// TIA Portal V17 export
// export: Created 2023-02-26T22:59:49.7304626Z, ExportSetting WithDefaults, DisplayName Totally Integrated Automation Portal, DisplayVersion V17, DisplayName TIA Portal Openness, DisplayVersion V17, DisplayName TIA Portal Version Control Interface, DisplayVersion V17, DisplayName TIA Portal Test Suite Advanced, DisplayVersion V17, DisplayName STEP 7 Professional, DisplayVersion V17, DisplayName SIMATIC Energy Suite, DisplayVersion V17, DisplayName STEP 7 Safety, DisplayVersion V17, DisplayName WinCC Professional, DisplayVersion V17
FUNCTION "LOG_ModeTime" : Void   // FC18, LAD
{ S7_Optimized_Access := 'TRUE' }
VERSION : 0.1
// stored: AutoNumber true, IsIECCheckEnabled false, SetENOAutomatically false, UDAEnableTagReadback false
   VAR_TEMP
      t_RisingEdge : Bool;
   END_VAR
BEGIN

REGION Network 1: Trigger
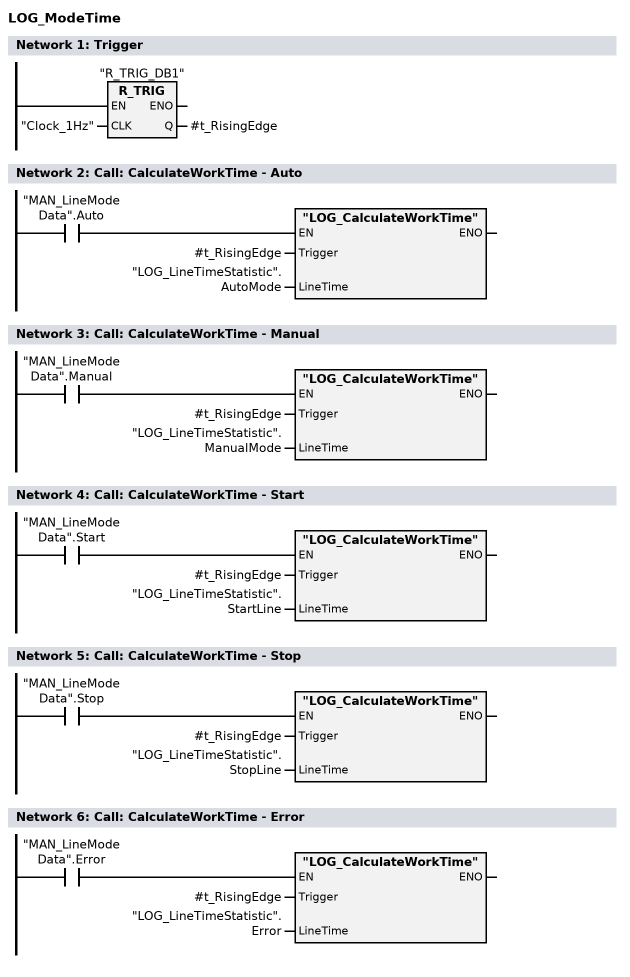
   RUNG wire#powerrail
      "R_TRIG_DB1".R_TRIG(CLK := "Clock_1Hz", Q => #t_RisingEdge)
   END_RUNG
   // the same network as SCL:
   "R_TRIG_DB1"(CLK := "Clock_1Hz", Q => #t_RisingEdge);   // R_TRIG
END_REGION

REGION Network 2: Call: CalculateWorkTime - Auto
   RUNG wire#powerrail
      Contact( "MAN_LineModeData".Auto )
      "LOG_CalculateWorkTime"(Trigger := #t_RisingEdge, LineTime := "LOG_LineTimeStatistic".AutoMode)
   END_RUNG
   // the same network as SCL:
   IF "MAN_LineModeData".Auto THEN
       "LOG_CalculateWorkTime"(Trigger := #t_RisingEdge, LineTime := "LOG_LineTimeStatistic".AutoMode);
   END_IF;
END_REGION

REGION Network 3: Call: CalculateWorkTime - Manual
   RUNG wire#powerrail
      Contact( "MAN_LineModeData".Manual )
      "LOG_CalculateWorkTime"(Trigger := #t_RisingEdge, LineTime := "LOG_LineTimeStatistic".ManualMode)
   END_RUNG
   // the same network as SCL:
   IF "MAN_LineModeData".Manual THEN
       "LOG_CalculateWorkTime"(Trigger := #t_RisingEdge, LineTime := "LOG_LineTimeStatistic".ManualMode);
   END_IF;
END_REGION

REGION Network 4: Call: CalculateWorkTime - Start
   RUNG wire#powerrail
      Contact( "MAN_LineModeData".Start )
      "LOG_CalculateWorkTime"(Trigger := #t_RisingEdge, LineTime := "LOG_LineTimeStatistic".StartLine)
   END_RUNG
   // the same network as SCL:
   IF "MAN_LineModeData".Start THEN
       "LOG_CalculateWorkTime"(Trigger := #t_RisingEdge, LineTime := "LOG_LineTimeStatistic".StartLine);
   END_IF;
END_REGION

REGION Network 5: Call: CalculateWorkTime - Stop
   RUNG wire#powerrail
      Contact( "MAN_LineModeData".Stop )
      "LOG_CalculateWorkTime"(Trigger := #t_RisingEdge, LineTime := "LOG_LineTimeStatistic".StopLine)
   END_RUNG
   // the same network as SCL:
   IF "MAN_LineModeData".Stop THEN
       "LOG_CalculateWorkTime"(Trigger := #t_RisingEdge, LineTime := "LOG_LineTimeStatistic".StopLine);
   END_IF;
END_REGION

REGION Network 6: Call: CalculateWorkTime - Error
   RUNG wire#powerrail
      Contact( "MAN_LineModeData".Error )
      "LOG_CalculateWorkTime"(Trigger := #t_RisingEdge, LineTime := "LOG_LineTimeStatistic".Error)
   END_RUNG
   // the same network as SCL:
   IF "MAN_LineModeData".Error THEN
       "LOG_CalculateWorkTime"(Trigger := #t_RisingEdge, LineTime := "LOG_LineTimeStatistic".Error);
   END_IF;
END_REGION
END_FUNCTION
